FUNCTION myfmod : LREAL
VAR_INPUT
	x,y:LREAL;
END_VAR
VAR
END_VAR

myfmod:=x-floor(x/y)*y;

END_FUNCTION

(* stored: Version 1.1.0.1, ProductVersion 3.1.4024.12
   POU myfmod: Id {a0b56290-3c9e-4706-85fe-f22bd031e29e}, SpecialFunc None *)
